// Mitsubishi GX Works2 project: Tap2V1FX3U   PLC: FX3U/FX3UC

// global labels: Global1
VAR_GLOBAL
  YYLimitN AT M8354 : BOOL;
  YYLimitP AT M8353 : BOOL;
  YYBusy AT M8350 : BOOL;
  YYInterruptInverse AT M8357 : BOOL;
  YYPos AT D8350 : DINT;
  YYAccelTime AT D8358 : INT;
  YYDecelTime AT D8359 : INT;
  YYPosView AT D0 : DINT;
  YYTarPos AT D2 : DINT;
  YYFeed AT D4 : DINT;
  YYPPM AT D6 : DINT;
  YYTarR AT M0 : BOOL;
  YYTarRSkip AT D8 : INT;
  YYOn AT M1 : BOOL;
  YYRun AT M2 : BOOL;
  YYDirection AT M3 : BOOL;
  YYReady AT M4 : BOOL;
  YYReadyI AT X005 : BOOL;
  YYPulseO AT Y001 : BOOL;
  YYDirectionO AT Y005 : BOOL;
  YYOnO AT Y011 : BOOL;
  YYInTorqueI AT X011 : BOOL;
  YYInTorqueIEdge AT M5 : BOOL;
  YYOverTorque AT M6 : BOOL;
  ZZLimitN AT M8364 : BOOL;
  ZZLimitP AT M8363 : BOOL;
  ZZBusy AT M8360 : BOOL;
  ZZInterruptInverse AT M8367 : BOOL;
  ZZPos AT D8360 : DINT;
  ZZAccelTime AT D8368 : INT;
  ZZDecelTime AT D8369 : INT;
  ZZPosView AT D9 : DINT;
  ZZTarPos AT D11 : DINT;
  ZZFeed AT D13 : DINT;
  ZZPPR AT D15 : DINT;
  ZZTarR AT M7 : BOOL;
  ZZTarRSkip AT D17 : INT;
  ZZRun AT M8 : BOOL;
  ZZDirection AT M9 : BOOL;
  ZZReadyI AT X006 : BOOL;
  ZZPulseO AT Y002 : BOOL;
  ZZDirectionO AT Y006 : BOOL;
  ZZOnO AT Y012 : BOOL;
  ZZInTorqueI AT X012 : BOOL;
  ZZInTorqueIEdge AT M10 : BOOL;
  ZZOverTorque AT M11 : BOOL;
  RunState AT D18 : INT;
  RunStateNext AT M12 : BOOL;
  AxisTapState AT D19 : INT;
  AxisTapStateNext AT M13 : BOOL;
  FoilExtractState AT D20 : INT;
  FoilExtractStateNext AT M14 : BOOL;
  FoilClampState AT D21 : INT;
  FoilClampStateNext AT M15 : BOOL;
  FoilSupplyState AT D22 : INT;
  FoilSupplyStateNext AT M16 : BOOL;
  FoilExtractDropN AT M17 : BOOL;
  FoilExtractDropNTimer AT TC0 : BOOL;
  FoilExtractDropNTimerDelay AT D23 : INT;
  FoilExtractDropP AT M18 : BOOL;
  FoilExtractDropPTimer AT TC1 : BOOL;
  FoilExtractDropPTimerDelay AT D24 : INT;
  FoilExtractDrop AT M19 : BOOL;
  FoilExtractDropO AT Y000 : BOOL;
  FoilClampN AT M20 : BOOL;
  FoilClampNTimer AT TC2 : BOOL;
  FoilClampNTimerDelay AT D25 : INT;
  FoilClampP AT M21 : BOOL;
  FoilClampPTimer AT TC3 : BOOL;
  FoilClampPTimerDelay AT D26 : INT;
  FoilClampPI AT X000 : BOOL;
  FoilClamp AT M22 : BOOL;
  FoilClampO AT Y003 : BOOL;
  FoilSupply AT M23 : BOOL;
  FoilSupplyO AT Y004 : BOOL;
  WorkFeedSpin AT D27 : DINT;
  WorkFeedTapTravelFast AT D29 : DINT;
  WorkFeedTapSpinForward AT D31 : DINT;
  WorkFeedTapSpinBack AT D33 : DINT;
  FoilFull AT M24 : BOOL;
  FoilFullI AT X001 : BOOL;
  FoilFullTimer AT TC4 : BOOL;
  AirReady AT M25 : BOOL;
  AirReadyI AT X002 : BOOL;
  Run AT M26 : BOOL;
  RunI AT X003 : BOOL;
  RunStop AT M27 : BOOL;
  RunStopI AT X004 : BOOL;
  SettingTapPitch AT D35 : DINT;
  SettingTapPitchI AT X007 : BOOL;
  SettingFoilSupplyI AT X010 : BOOL;
  SettingTapSpinSpeedI AT X013 : BOOL;
  SettingTapTravelBegin AT D37 : DINT;
  SettingTapTravelEnd AT D39 : DINT;
  TapMoveToTravelBegin AT M28 : BOOL;
  TapCount AT D41 : DINT;
  TapCountAtSupplyEnd AT D43 : DINT;
  StopTap AT M29 : BOOL;
  StopTapTimer AT TC5 : BOOL;
  StopClamp AT M30 : BOOL;
  StopClampPLS AT M31 : BOOL;
  StopClampTimer AT TC6 : BOOL;
  Alert AT M32 : BOOL;
  AlertTimer AT TC7 : BOOL;
  AlertO AT Y007 : BOOL;
  ErrorReset AT M33 : BOOL;
  ErrorResetTimer AT TC8 : BOOL;
  ErrorResetO AT Y010 : BOOL;
  Overload AT M34 : BOOL;
END_VAR

// task Task_01 (event TRUE, interval 0, priority 31): POU_01

PROGRAM POU_01
VAR
  fTmp : BOOL;
END_VAR
RST(M8002, YYOn);
MOV(M8002, 100, YYAccelTime); MOV(M8002, YYAccelTime, ZZAccelTime);
MOV(M8002, 100, YYDecelTime); MOV(M8002, YYDecelTime, ZZDecelTime);
RST(M8002, YYOverTorque);
RST(M8002, ZZOverTorque);
RST(M8002, FoilExtractDrop);
RST(M8002, FoilClamp);
RST(M8002, FoilSupply);
SET(M8002, Alert);
(*y axis: tap travel*)
DMOV(M8002, 1_000, YYPPM);
RST(M8002, TapCount);
DMOV(M8002, 100_000, WorkFeedTapTravelFast);
(*z axis: tap spin*)
DMOV(M8002, YYPPM, ZZPPR);
(*it easier to calculate if YYPPM = ZZPPR*)
(*|||||||||||||||*)

(*|||||||||||||||*)
SET(Run AND RunState = 0 AND AirReady, fTmp);
RST(fTmp, Run);
SET(fTmp, YYOn);
SET(fTmp, TapMoveToTravelBegin);
RST(fTmp, StopClamp);
MOV(fTmp, 1, RunState);
RST(fTmp, fTmp);
SET(RunStop OR Overload, fTmp);
SET(fTmp AND RunStop, ErrorReset);
RST(fTmp, Run);
RST(fTmp, RunStop);
RST(fTmp, Overload);
SET(fTmp, Alert);
ZRST(fTmp, RunState, FoilSupplyState);
RST(fTmp, YYRun);
RST(fTmp, ZZRun);
SET(fTmp AND YYOn, StopTap);
RST(fTmp, FoilExtractDrop);
RST(fTmp, FoilClamp);
RST(fTmp, FoilSupply);
RST(fTmp, fTmp);
OUT_T(StopTap, StopTapTimer, 5);
RST(StopTapTimer, YYOn);
RST(StopTapTimer, StopTap);

(*|||||||||||||||*)
(*|||||||||||||||*)
INC(RunStateNext, RunState);
INC(AxisTapStateNext, AxisTapState);
INC(FoilExtractStateNext, FoilExtractState);
INC(FoilClampStateNext, FoilClampState);
INC(FoilSupplyStateNext, FoilSupplyState);
ZRST(M8000, RunStateNext, FoilSupplyStateNext);
DECO(M8000, RunState, 6, M100);
DECO(M8000, AxisTapState, 6, M200); DECO(M8000, AxisTapState, 6, M1200); ZRST(NOT YYReady, M1200, M1263);
DECO(M8000, FoilExtractState, 6, M300);
DECO(M8000, FoilClampState, 6, M400);
DECO(M8000, FoilSupplyState, 6, M500);
(*|||||||||||||||*)

(*|||||||||||||||*)
(*origin tap, extract, clamp, supply*)
MOV(M101, 1, AxisTapState);
MOV(M101, 1, FoilExtractState);
MOV(M101, 1, FoilClampState);
MOV(M101, 1, FoilSupplyState);
DMOV(M101, TapCount - 8, TapCountAtSupplyEnd);
SET(M101, RunStateNext);
(*ready done, run command -> cycle start*)
SET(M102 AND M1220 AND M320 AND M420 AND Run, RunStateNext);
(*cycle start*)
SET(M103 AND M1220 AND M320 AND M420, fTmp);
SET(fTmp, Alert);
SET(fTmp, RunStateNext);
RST(fTmp, fTmp);
(*foil extract drop*)
MOV(M104, 11, FoilExtractState);
SET(M104, RunStateNext);
(*foil extract drop done -> clamp on*)
MOV(M105 AND M315, 11, FoilClampState);
SET(M105 AND M315, RunStateNext);
(*clamp on done -> tap, foil extract block*)
SET(M106 AND M415, fTmp);
MOV(fTmp, 11, AxisTapState);
MOV(fTmp, 16, FoilExtractState);
MOV(fTmp, 11, RunState);
RST(fTmp, fTmp);
(*tap done, foil extract block done -> clamp off, add tap count*)
SET(M111 AND M1220 AND M320, fTmp);
MOV(fTmp, 16, FoilClampState);
DINC(fTmp, TapCount);
SET(fTmp, RunStateNext);
RST(fTmp, fTmp);
(*clamp off done -> return cycle start*)
SET(M112 AND M420, fTmp);
MOV(fTmp, 3, RunState);
RST(fTmp, Alert);
RST(fTmp, fTmp);
(*|||||||||||||||*)
(*foil full -> record*)
DMOV(FoilFull, TapCount, TapCountAtSupplyEnd);
(*check*)
SET((TapCount - TapCountAtSupplyEnd) >= 8, fTmp);
RST(NOT SettingFoilSupplyI, fTmp);
OUT(fTmp AND NOT FoilFull AND M520, FoilSupply);
RST(fTmp, fTmp);
(*|||||||||||||||*)

(*|||||||||||||||*)
(*/////get origin tap*)
(*move back*)
SET(M1201, fTmp);
RST(fTmp, YYPos); RST(fTmp, ZZPos);
DMOV(fTmp, -100_000, YYTarPos); DMOV(fTmp, YYTarPos * ZZPPR / SettingTapPitch, ZZTarPos);
DMOV(fTmp, 5_000, YYFeed); DMOV(fTmp, YYFeed * ZZPPR / SettingTapPitch, ZZFeed);
SET(fTmp, YYRun); SET(fTmp, ZZRun);
SET(fTmp, AxisTapStateNext);
RST(fTmp, fTmp);
(*move back hit hard limit -> reset*)
SET(M202 AND NOT YYBusy, fTmp);
RST(fTmp, YYRun); RST(fTmp, ZZRun);
RST(fTmp, YYPos); RST(fTmp, ZZPos);
SET(fTmp, AxisTapStateNext);
RST(fTmp, fTmp);
(*move forward*)
SET(M1203, fTmp);
DMOV(fTmp, 5_000, YYTarPos);
DMOV(fTmp, 1_000, YYFeed);
SET(fTmp, YYRun);
SET(fTmp, AxisTapStateNext);
RST(fTmp, fTmp);
(*move forward out limit, stop*)
SET(M204 AND YYInTorqueI, fTmp);
RST(fTmp, YYRun);
SET(fTmp, AxisTapStateNext);
RST(fTmp, fTmp);
(*stop done, move forward x mm*)
SET(M1205, fTmp);
DMOV(fTmp, YYPos + 1_000, YYTarPos);
DMOV(fTmp, 5_000, YYFeed);
SET(fTmp, YYRun);
SET(fTmp, AxisTapStateNext);
RST(fTmp, fTmp);
(*move forward x mm done -> reset, move to begin or end*)
SET(M1206, fTmp);
RST(fTmp, YYPos); RST(fTmp, ZZPos);
MOV(fTmp AND TapMoveToTravelBegin, 7, AxisTapState);
MOV(fTmp AND NOT TapMoveToTravelBegin, 8, AxisTapState);
RST(fTmp, fTmp);
(*move to begin*)
DMOV(M1207, SettingTapTravelBegin, YYTarPos);
DMOV(M1207, 20_000, YYFeed);
SET(M1207, YYRun);
SET(M1207, AxisTapStateNext);
(*ready*)
MOV(M1208, 20, AxisTapState);
(*/////main sequence*)
(*move forward*)
SET(M1211, fTmp);
DMOV(fTmp, SettingTapTravelEnd, YYTarPos); RST(fTmp, ZZPos); DMOV(fTmp, (YYTarPos - YYPos) * ZZPPR / SettingTapPitch, ZZTarPos);
DMOV(fTmp, WorkFeedTapSpinForward, ZZFeed); DMOV(fTmp, ZZFeed * SettingTapPitch / ZZPPR, YYFeed);
SET(fTmp, YYRun); SET(fTmp, ZZRun);
SET(fTmp, AxisTapStateNext); RST(fTmp, fTmp);
(*move forward done -> back lash eliminate*)
DMOV(M1212, SettingTapTravelEnd - 0_020, YYTarPos);
DMOV(M1212, 2_000, YYFeed);
SET(M1212, YYRun);
SET(M1212, AxisTapStateNext);
(*backlash eliminate done -> move back*)
SET(M1213, fTmp);
DMOV(fTmp, SettingTapTravelBegin, YYTarPos); RST(fTmp, ZZPos); DMOV(fTmp, (YYTarPos - YYPos) * ZZPPR / SettingTapPitch, ZZTarPos);
DMOV(fTmp, WorkFeedTapSpinBack, ZZFeed); DMOV(fTmp, ZZFeed * SettingTapPitch / ZZPPR, YYFeed);
SET(fTmp, YYRun); SET(fTmp, ZZRun);
SET(fTmp, AxisTapStateNext); RST(fTmp, fTmp);
(*move back done -> end*)
SET(M1214, fTmp);
MOV(fTmp, 20, AxisTapState); RST(fTmp, fTmp);
(*|||||||||||||||*)

(*|||||||||||||||*)
(*/////get origin foil extract*)
(*drop back*)
RST(M301, FoilExtractDrop);
SET(M301, FoilExtractStateNext);
(*drop back done -> next*)
SET(M302 AND FoilExtractDropN, FoilExtractStateNext);
(*end*)
MOV(M303, 20, FoilExtractState);
(*/////drop*)
(*drop forward*)
SET(M311, FoilExtractDrop);
SET(M311, FoilExtractStateNext);
(*drop forward done*)
MOV(M312 AND FoilExtractDropP, 15, FoilExtractState);
(*/////block*)
(*drop back*)
RST(M316, FoilExtractDrop);
SET(M316, FoilExtractStateNext);
(*drop back done*)
MOV(M317 AND FoilExtractDropN, 20, FoilExtractState);
(*|||||||||||||||*)

(*|||||||||||||||*)
(*/////get origin foil clamp*)
(*back*)
RST(M401, FoilClamp);
SET(M401, FoilClampStateNext);
(*back done -> next*)
SET(M402 AND FoilClampN, FoilClampStateNext);
(*end*)
MOV(M403, 20, FoilClampState);
(*/////clamp on*)
(*forward*)
SET(M411, FoilClamp);
SET(M411, FoilClampStateNext);
(*forward done -> done*)
MOV(M412 AND FoilClampP, 15, FoilClampState);
(*/////clamp off*)
(*back*)
RST(M416, FoilClamp);
SET(M416, FoilClampStateNext);
(*back done -> done*)
MOV(M417 AND FoilClampN, 20, FoilClampState);
(*|||||||||||||||*)

(*|||||||||||||||*)
(*/////get origin foil supply*)
(*reset*)
RST(M501, FoilSupply);
SET(M501, FoilSupplyStateNext);
(*end*)
MOV(M502, 20, FoilSupplyState);
(*/////supply sequence*)
(*|||||||||||||||*)

(*|||||||||||||||*)
(*YY*)
RST(YYRun AND YYTarPos = YYPos, YYRun);
DDRVA(YYRun, YYTarPos, YYFeed, YYPulseO, YYDirection);
RST(M8029, YYRun);
OUT(NOT YYDirection, YYDirectionO);
INC(NOT YYRun AND NOT YYBusy AND YYTarRSkip < 5, YYTarRSkip);
RST(YYRun, YYTarRSkip);
OUT(YYTarRSkip >= 5, YYTarR);
(*|||||||||||||||*)
(*ZZ*)
RST(ZZRun AND ZZTarPos = ZZPos, ZZRun);
DDRVA(ZZRun, ZZTarPos, ZZFeed, ZZPulseO, ZZDirection);
RST(M8029, ZZRun);
OUT(NOT ZZDirection, ZZDirectionO);
INC(NOT ZZRun AND NOT ZZBusy AND ZZTarRSkip < 5, ZZTarRSkip);
RST(ZZRun, ZZTarRSkip);
OUT(ZZTarRSkip >= 5, ZZTarR);
(*|||||||||||||||*)
(*ready*)
OUT(YYReadyI AND YYTarR AND ZZReadyI AND ZZTarR, YYReady);
(*limit*)
OUT(NOT YYDirection AND NOT YYInTorqueI, YYLimitN); OUT(YYLimitN, ZZLimitN);
(*|||||||||||||||*)

(*|||||||||||||||*)
PLS(RunI, Run); SET(Run, Run);
PLF(RunStopI, RunStop); SET(RunStop, RunStop);
OUT_T(NOT RunStopI AND NOT StopClamp, StopClampTimer, 20); SET(StopClampTimer, StopClamp);
RST(StopClamp, RunStop);
SET(StopClamp, FoilClamp);
SET(StopClamp AND FoilClampP, fTmp);
SET(fTmp, YYOn);
MOV(fTmp, 1, AxisTapState);
RST(fTmp, StopClamp);
RST(fTmp, TapMoveToTravelBegin);
RST(fTmp, fTmp);
PLF(YYInTorqueI, YYInTorqueIEdge); SET(YYInTorqueIEdge, YYOverTorque); SET(YYInTorqueIEdge AND YYDirection, Overload);
PLS(ZZInTorqueI, ZZInTorqueIEdge); SET(ZZInTorqueIEdge, ZZOverTorque); SET(ZZInTorqueIEdge, Overload);
(*foil extract*)
MOV(M8002, 5, FoilExtractDropNTimerDelay);
OUT_T(NOT FoilExtractDrop, FoilExtractDropNTimer, FoilExtractDropNTimerDelay); SET(FoilExtractDropNTimer, FoilExtractDropN); RST(FoilExtractDropNTimer, FoilExtractDropP);
MOV(M8002, 5, FoilExtractDropPTimerDelay);
OUT_T(FoilExtractDrop, FoilExtractDropPTimer, FoilExtractDropPTimerDelay); SET(FoilExtractDropPTimer, FoilExtractDropP); RST(FoilExtractDropPTimer, FoilExtractDropN);
(*foil clamp*)
MOV(M8002, 3, FoilClampNTimerDelay);
OUT_T(NOT FoilClamp AND NOT FoilClampPI, FoilClampNTimer, FoilClampNTimerDelay); SET(FoilClampNTimer, FoilClampN); RST(FoilClampNTimer, FoilClampP);
MOV(M8002, 3, FoilClampPTimerDelay);
OUT_T(FoilClamp AND FoilClampPI, FoilClampPTimer, FoilClampPTimerDelay); SET(FoilClampPTimer, FoilClampP); RST(FoilClampPTimer, FoilClampN);
(*foil supply*)
OUT_T(FoilFullI, FoilFullTimer, 8); OUT(FoilFullTimer, FoilFull);
(*setting pitch*)
DMOV(NOT SettingTapPitchI, 1_000, SettingTapPitch);
DMOV(SettingTapPitchI, 1_270, SettingTapPitch);
(*setting feed*)
DMOV(NOT SettingTapSpinSpeedI, (ZZPPR * 1_200) / 60, WorkFeedTapSpinForward);
DMOV(NOT SettingTapSpinSpeedI, (ZZPPR * 1_200) / 60, WorkFeedTapSpinBack);
DMOV(SettingTapSpinSpeedI, (ZZPPR * 1_400) / 60, WorkFeedTapSpinForward);
DMOV(SettingTapSpinSpeedI, (ZZPPR * 1_400) / 60, WorkFeedTapSpinBack);
(*setting travel*)
DMOV(M8002, 5_000, SettingTapTravelBegin);
DMOV(M8002, SettingTapTravelBegin + 25_000, SettingTapTravelEnd);
(**)
OUT(AirReadyI, AirReady);
(*|||||||||||||||*)
OUT(YYOn, YYOnO); OUT(YYOn, ZZOnO);
OUT(FoilExtractDrop, FoilExtractDropO);
OUT(FoilClamp, FoilClampO);
OUT(FoilSupply, FoilSupplyO);
OUT(AlertTimer, AlertO);
OUT(ErrorReset, ErrorResetO);
(**)
OUT_T(ErrorReset, ErrorResetTimer, 1); RST(ErrorResetTimer, ErrorReset);
RST(ErrorResetTimer, YYOverTorque);
RST(ErrorResetTimer, ZZOverTorque);
OUT_T(Alert, AlertTimer, 100);
(*|||||||||||||||*)
END_PROGRAM
